// SIMATIC S7-200 project (STEP 7-Micro/WIN), CPU 224XP REL 02.01

SYMBOL_TABLE 用户定义1
紧急启动             I1.1
急停保持原位           0
料钩反转             Q0.3
料钩正转             Q0.2
天车反转             Q0.1
天车正转             Q0.0     // 天车正转
原点下降             M1.6     // 料钩反转
后退原点             I0.7
二号后退             M1.5     // 送料天车正转
二号上升             M1.4     // 料钩正转
一百秒              T41      // 清洗100s
二号清洗             M1.3
二号下降             M1.2     // 料钩反转
二号到位             I0.6
一号后退             M1.1     // 送料天车正转
一号上升             M1.0     // 料钩正转
二百秒              T40      // 一号电镀200s
一号电镀             M2.7
一号下降             M2.6     // 料钩反转
一号到位             I0.5
零号后退             M2.5     // 送料天车正转
零号上升             M2.4     // 料钩正转
三百秒              T39      // 0号电镀300s
零号电镀             M2.3
下限位              I0.4
零号下降             M2.2     // 料钩反转
零号到位             I0.3
前进               M2.1     // 送料天车反转
原点上升             M2.0     // 料钩正转
上限位              I0.2
qidong           I0.0     // 启动
暂停               I0.1     // 暂停
END_SYMBOL_TABLE

ORGANIZATION_BLOCK 主程序:OB1
TITLE=【PLC一条电泳线流水线控制程序实例】
// 程序运行时，首先按下启动按钮，若紧急启动按钮未触发，原点上升控制置位，驱动料钩正转输出使料钩上升。在启动料钩上升前，系统应检查上限位传感器是否未触发，以防设备因过度上升受损。料钩升至合适高度后，前进控制激活天车反转输出，将工件送至零号工位。当零号到位传感器触发，零号下降控制置位，驱动料钩反转输出使料钩下降，直至下限位传感器确认到位。随后，零号电镀控制启动三百秒定时器，进行300秒电镀。在启动三百秒定时器前，系统需确认下限位传感器已触发，以确保电镀质量。电镀完成后，零号上升控制再次驱动料钩正转输出，料钩上升，零号后退控制激活天车正转输出，工件被送往下一工位。
// 在一号工位，一号到位传感器触发后，一号下降控制使料钩下降，下降到位后一号电镀控制启动二百秒定时器，进行200秒电镀。在启动二百秒定时器前，系统需确认下限位传感器已触发。之后，一号上升控制和一号后退控制依次执行，工件被送至二号工位。二号到位传感器触发后，二号下降控制使料钩下降，二号清洗控制启动一百秒定时器清洗100秒。在启动一百秒定时器前，系统需确认下限位传感器已触发。清洗结束，二号上升控制提升料钩，二号后退控制驱动天车正转输出，工件回到原点，后退原点传感器触发后，原点下降控制完成最后下降。
// 系统确保料钩正转输出和料钩反转输出不同时激活，以避免电机冲突；同样，系统确保天车正转输出和天车反转输出不同时激活，以防止驱动系统损坏。若暂停按钮按下，系统暂停当前操作；当紧急启动按钮触发时，系统立即停止所有输出，确保安全。
// 
BEGIN
Network 1
LD     qidong:I0.0
EU
AW=    MW1, 急停保持原位
O      原点上升:M2.0
LPS
AN     前进:M2.1
=      原点上升:M2.0
LPP
R      M1.7, 1
Network 2
LD     qidong:I0.0
A      紧急启动:I1.1
O      原点上升:M2.0
AN     暂停:I0.1
MOVW   1, MW3
Network 3
LD     暂停:I0.1
MOVW   3, MW3
Network 4
LDW=   MW3, 1
=      M30.0
Network 5
LD     上限位:I0.2
A      原点上升:M2.0
LD     零号到位:I0.3
A      前进:M2.1
OLD
LD     下限位:I0.4
A      零号下降:M2.2
OLD
LD     三百秒:T39
A      零号电镀:M2.3
OLD
LD     上限位:I0.2
A      零号上升:M2.4
OLD
LD     一号到位:I0.5
A      零号后退:M2.5
OLD
LD     下限位:I0.4
A      一号下降:M2.6
OLD
LD     二百秒:T40
A      一号电镀:M2.7
OLD
LD     上限位:I0.2
A      一号上升:M1.0
OLD
LD     二号到位:I0.6
A      一号后退:M1.1
OLD
LD     下限位:I0.4
A      二号下降:M1.2
OLD
LD     一百秒:T41
A      二号清洗:M1.3
OLD
LD     上限位:I0.2
A      二号上升:M1.4
OLD
LD     后退原点:I0.7
A      二号后退:M1.5
OLD
LD     下限位:I0.4
A      原点下降:M1.6
OLD
AN     M1.7
EU
A      M30.0
SLW    MW1, 1
Network 6
LD     零号电镀:M2.3
TON    三百秒:T39, 300
Network 7
LD     一号电镀:M2.7
TON    二百秒:T40, 200
Network 8
LD     二号清洗:M1.3
TON    一百秒:T41, 100
Network 9
LD     零号后退:M2.5
O      一号后退:M1.1
O      二号后退:M1.5
A      M30.0
=      天车正转:Q0.0
Network 10
LD     前进:M2.1
A      M30.0
=      天车反转:Q0.1
Network 11
LD     二号上升:M1.4
O      零号上升:M2.4
O      一号上升:M1.0
O      原点上升:M2.0
A      M30.0
=      料钩正转:Q0.2
Network 12
LD     零号下降:M2.2
O      一号下降:M2.6
O      二号下降:M1.2
O      原点下降:M1.6
A      M30.0
=      料钩反转:Q0.3
END_ORGANIZATION_BLOCK
